{attribute addProperty BoxType "EL6001-0000-0017"}
{attribute addProperty Id "COM_InputsAT %I*COM_Inputs_85D1D733192240COM_OutputsAT %Q*COM_Outputs_AC29F8FC192240WcStateAT %I*WcState_F855686C1620InfoDataAT %I*InfoData_BC63D37F80100"}
{attribute addProperty CRC "2580370976"}
{attribute addProperty SizeInBites "480"}
{attribute addProperty SizeInBytes "60"}
TYPE EL6001_5D31AA51 :
STRUCT
	{attribute addProperty Name "COM_Inputs"}
	COM_Inputs : COM_Inputs_85D1D733;
	{attribute addProperty Name "COM_Outputs"}
	COM_Outputs : COM_Outputs_AC29F8FC;
	{attribute addProperty Name "WcState"}
	WcState : WcState_F855686C;
	{attribute addProperty Name "InfoData"}
	InfoData : InfoData_BC63D37F;
END_STRUCT
END_TYPE

(* stored: Version 1.2.0.0, ProductVersion 3.1.4024.9
   DUT EL6001_5D31AA51: Id {33ddab99-63ba-4a6c-a1a7-347cd237c579} *)
